{attribute 'pack_mode' := '1'}  // needed for python pyads reading
TYPE ST_ManMov_FreeMove :
STRUCT
	move_position_CMD_enable:BOOL;
	move_position_CMD_done: BOOL;
	move_position :MoverVector;
END_STRUCT
END_TYPE

(* stored: Version 1.1.0.1
   DUT ST_ManMov_FreeMove: Id {e999d679-fde2-4260-917e-710d19ca26ab} *)
